// TIA Portal V18 export
TYPE "KISTLER_HMI_DATA"
// stored: IsFailsafeCompliant false
   STRUCT
      PRESS_ID : Int;
      Enable : Bool;
      Home_set : Bool;
      Home_End : Bool;
      REF_Set : Bool;
      REF_End : Bool;
      SELECT_PROGRAM : Bool;
      SELECT_PRO_End : Bool;
      SYS_Alarm : Bool;
      SYS_Ready : Bool;
      Cyc_Start : Bool;
      Cyc_Start_OK : Bool;
      Cyc_Start_Nok : Bool;
      Press_Result_OK : Bool;
      Press_Result_NG : Bool;
      "JOG+" : Bool;
      "JOG-" : Bool;
      "Force actual" : Real;
      "Position actual" : Real;
      Write_PRO_ID : Byte;
      Read_PRO_ID : Byte;
      servoJogSpeed : Real;
      ServoManualMaxForce : Real;
      Write_Data : Bool;
      Write_Data_End : Bool;
      Write_Data_Alarm : Bool;
      "Position actual_1" : Real;
      Out_UNI_0 : Bool;
      IN_UNI_0 : Bool;
      DisableEnable : Bool;
      EnableState : Bool;
   END_STRUCT;
END_TYPE
